(* IEC 61131-3 sources: CodesysTest/alpha/export/FBs/Components/DelayDwellFB/DelayDwellFB.pou, 1 file *)

(* ---- Reset.m.st ---- *)
(*#-#-#-#-#-#-#-#-#-#---Declaration---#-#-#-#-#-#-#-#-#-#-#-#-#*)

METHOD Reset : BOOL
VAR_INPUT
END_VAR
(*#-#-#-#-#-#-#-#-#-#---Implementation---#-#-#-#-#-#-#-#-#-#-#-#-#*)

active := FALSE;
_trigger := FALSE;
_manualOn := FALSE;
_manualOff := FALSE;
Q := FALSE;
state := DELAY_DWELL_STATES.Idle;
